{attribute 'linkalways'} 
{attribute 'no_explicit_call' := 'This FB is a CLASS and must be accessed using methods or properties'}
{attribute 'enable_dynamic_creation'}
FUNCTION_BLOCK ChunkedRequestData EXTENDS Disposable IMPLEMENTS I_ChunkedRequestData
VAR
	maximumChunkSizeInBytes : UDINT;
	totalReceivedChunks : UDINT;
	totalExpectedChunks : UDINT;
	pPayloadBuffer : POINTER TO STRING;
	payloadBufferSize : UDINT;
END_VAR

METHOD PRIVATE CreateBuffer
VAR_INPUT
	SizeInBytes : UDINT;
END_VAR
payloadBufferSize := SizeInBytes;
pPayloadBuffer := __NEW(BYTE, SizeInBytes);
memset(pPayloadBuffer, 0, SizeInBytes);
END_METHOD

METHOD PRIVATE DestroyBuffer
VAR_INPUT
END_VAR
IF pPayloadBuffer = 0 THEN
	RETURN;
END_IF

__DELETE(pPayloadBuffer);
pPayloadBuffer := 0;
END_METHOD

METHOD FB_exit : BOOL
VAR_INPUT
	bInCopyCode : BOOL; // if TRUE, the exit method is called for exiting an instance that is copied afterwards (online change).
END_VAR
IF bInCopyCode THEN
	RETURN;
END_IF

DestroyBuffer();
END_METHOD

METHOD FB_init : BOOL
VAR_INPUT
	bInitRetains : BOOL; // if TRUE, the retain variables are initialized (warm start / cold start)
	bInCopyCode : BOOL;  // if TRUE, the instance afterwards gets moved into the copy code (online change)
	ChunkSizeInBytes : UDINT;
	ChunkCount : UDINT;
END_VAR
maximumChunkSizeInBytes := ChunkSizeInBytes;
totalExpectedChunks := ChunkCount;
CreateBuffer(ChunkSizeInBytes * ChunkCount);
END_METHOD

PROPERTY PUBLIC IsComplete : BOOL
GET
IsComplete := totalReceivedChunks = totalExpectedChunks;
END_GET
END_PROPERTY

PROPERTY PUBLIC PayloadAddress : POINTER TO STRING
GET
PayloadAddress := pPayloadBuffer;
END_GET
END_PROPERTY

PROPERTY PUBLIC PayloadSizeInBytes : UDINT
GET
PayloadSizeInBytes := payloadBufferSize;
END_GET
END_PROPERTY

METHOD PUBLIC TryAddChunkedPayload : BOOL;
VAR_INPUT
	PayloadAddress : POINTER TO STRING;
	PayloadSize : UDINT;
	ChunkSequence : DINT;
END_VAR
VAR
	offset : UDINT;
	pBufferChunkLocation : POINTER TO BYTE;
END_VAR
IF totalReceivedChunks >= totalExpectedChunks THEN
	RETURN;
END_IF

IF PayloadSize > maximumChunkSizeInBytes THEN
	RETURN;
END_IF

IF ChunkSequence <= 0 THEN
	RETURN;
END_IF

concat2(pPayloadBuffer, PayloadAddress, pPayloadBuffer, payloadBufferSize);
totalReceivedChunks := totalReceivedChunks + 1;

TryAddChunkedPayload := TRUE;
END_METHOD

END_FUNCTION_BLOCK

(* stored: Version 1.1.0.1, ProductVersion 3.1.4024.13
   POU ChunkedRequestData: Id {7f5881bf-8a05-0b27-0aed-d7991d25f607}, SpecialFunc None
   Folder Constructor: Id {da25c027-5015-05bb-26a1-8f0167b8cc26}
   Folder Destructor: Id {611eebce-0bd8-05ea-20e8-f733449d4aac}
   Folder Private: Id {5dc5b110-b221-0389-0193-5300ad47d73e}
   Method CreateBuffer: Id {8996c178-6fd7-08dc-241e-865d4561c8b8}
   Method DestroyBuffer: Id {8e95d4e2-c36d-0403-14b6-2b3c556cc786}
   Method FB_exit: Id {fa1bb8f4-32ce-0721-26a6-bd31aa2e5062}
   Method FB_init: Id {7ca372bb-7a32-0bba-1d3e-9ca3233f191a}
   Property IsComplete: Id {b54c81e6-2980-0997-0ad6-4dc775a2e6e0}
   Get Get: Id {81b9c058-72bc-06b7-0425-c3bd424038a2}
   Property PayloadAddress: Id {fd5155a8-71ce-030c-3ccb-c20dce8c1414}
   Get Get: Id {c4fc4d05-ce0d-0410-0bb6-d484af2f2b92}
   Property PayloadSizeInBytes: Id {f9ff873e-6d8b-0c47-2996-a51051d7fb31}
   Get Get: Id {60cf9f56-a0a5-0f80-042a-7e0c41481657}
   Method TryAddChunkedPayload: Id {9fba7f24-853d-0cce-2be8-cc19d59d1bb2} *)
